TYPE ZONA_INPUT :
	STRUCT
		ENABLE     : BOOL;
		RIPRISTINO : BOOL;
		LIBERO     : BOOL;
		TRIGGER    : BOOL;
	END_STRUCT
END_TYPE

(* stored: Version 1.1.0.1, ProductVersion 3.1.4024.12
   DUT ZONA_INPUT: Id {26f55477-8a03-4053-8e7c-5088a18881a6} *)
